# EPICS StreamDevice protocol: serialTest/proto/client.proto
Terminator = CR LF;

request_data{
        out "\$1";
        in "%f";
}
